Staubli VAL3: deb230405.pjx

Parameters version=s7.4 stackSize=5000 millimeterUnit=true
Program file=deb.pgx
Program file=start.pgx
Program file=stop.pgx
Data file=deb230405.dtx
